Staubli VAL3: load.pgx

public program load(string x_sItem, num& x_nResult)
  local string l_sType
  local string l_sMessage
begin
  // load it

end
